TYPE stExternalCommand :
STRUCT
    SKILLID				: UINT;
	SKILLNAME			: STRING;
    bStart  : BOOL;
	bStop	: BOOL;
END_STRUCT
END_TYPE

(* stored: Version 1.1.0.1, ProductVersion 3.1.4026.18
   DUT stExternalCommand: Id {cad1bdb5-a271-4d06-8a47-25760d0f4170} *)
